FUNCTION alg_a: REAL
{ S7_Optimized_Access := 'false' }
    VAR_INPUT
        state: STATE;
    END_VAR

BEGIN
    alg_a := (state.cvar_c) + (derivcvar_c(state));
END_FUNCTION
